% RSLogix 500 project 002.RSS, saved by version 8.30.00.16 %
PROJECT "UNTITLED"    % processor: Bul.1763 MicroLogix 1100 Series B %

PROGRAM FILES
  LAD 2 "MAIN"  2 rungs
  LAD 3 "ALARMS"  1 rungs
  LAD 4 "IO"  3 rungs

DATA FILES
  O0 OUTPUT  5 elements
  I1 INPUT  7 elements
  S2 STATUS  66 elements
  B3 BINARY  1 elements
  T4 TIMER  1 elements
  C5 COUNTER  1 elements
  R6 CONTROL  1 elements
  N7 INTEGER  1 elements
  F8 FLOAT  1 elements

LADDER 2 "MAIN"
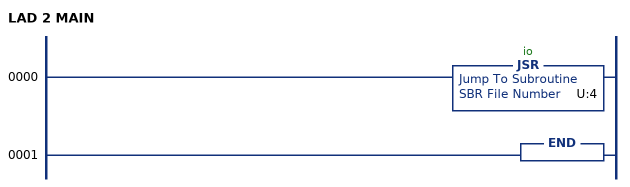
% Rung: 0 %  % edit flag set %
SOR JSR U:4 EOR
%   U:4  "io" %
% Rung: 1 %
SOR END EOR

LADDER 4 "IO"
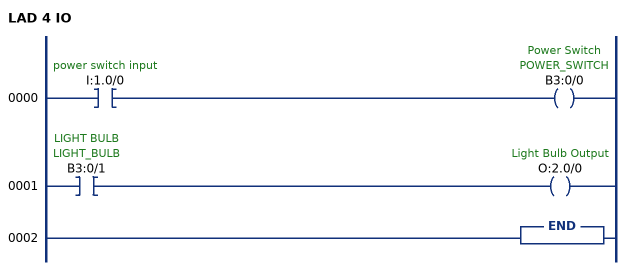
% Rung: 0 %
SOR XIC I:1.0/0 OTE B3:0/0 EOR
%   I:1.0/0  "power switch input" %
%   B3:0/0  POWER_SWITCH  "Power Switch" %
% Rung: 1 %
SOR XIC B3:0/1 OTE O:2.0/0 EOR
%   B3:0/1  LIGHT_BULB  "LIGHT BULB" %
%   O:2.0/0  "Light Bulb Output" %
% Rung: 2 %
SOR END EOR
